(* IEC 61131-3 sources: Industry-PLC-LLM/data/PLCBEAD_repo/PLCBEAD_PLCEmbed-main/PLC-BEAD/Source/GEB/OM_TO_F, 1 file *)

(* ---- OM_TO_F.ST ---- *)
FUNCTION OM_TO_F:REAL

	VAR_INPUT
		OM :	REAL;
	END_VAR

	OM_to_F := OM / 6.283185307179586476;

END_FUNCTION

PROGRAM program0
	VAR
		OM : REAL;
		OUT : REAL;
	END_VAR

	OUT := OM_TO_F(OM);
END_PROGRAM
